SUBAPPLICATION Versuch_405 (* Versuch Array Summe *)
  (* Standard: 61499-2; Description: Copyright (c) 2023 Meisterschulen am Ostbahnhof This program and the accompanying materials are made available under the terms of the Eclipse Public License 2.0 which is available at https://www.eclipse.org/legal/epl-2.0/ SPDX-License-Identifier: EPL-2.0 *)
  (* Version 1.0, 2023-10-23, Franz Höpfinger, Meisterschulen am Ostbahnhof *)
  PACKAGE Versuche;
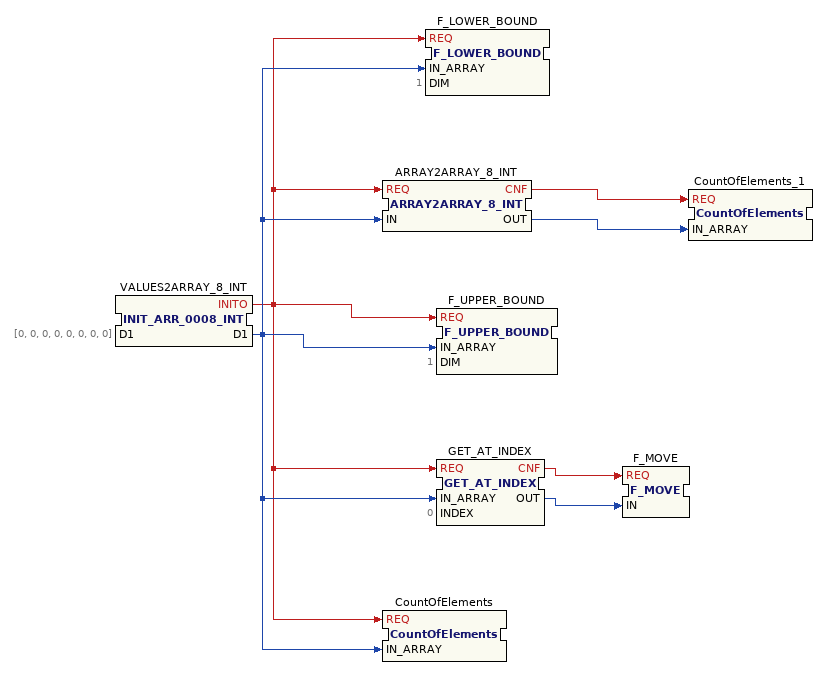
  FBS
    GET_AT_INDEX : eclipse4diac::convert::GET_AT_INDEX(INDEX := 0);
    F_MOVE : iec61131::selection::F_MOVE; {SET_ATTRIBUTE(DataType, INT)}
    CountOfElements : eclipse4diac::convert::CountOfElements;
    F_UPPER_BOUND : eclipse4diac::convert::F_UPPER_BOUND(DIM := 1);
    F_LOWER_BOUND : eclipse4diac::convert::F_LOWER_BOUND(DIM := 1);
    VALUES2ARRAY_8_INT : logiBUS::utils::generate::INIT_ARR_0008_INT(D1 := [0, 0, 0, 0, 0, 0, 0, 0]);
    ARRAY2ARRAY_8_INT : eclipse4diac::convert::ARRAY2ARRAY_8_INT;
    CountOfElements_1 : eclipse4diac::convert::CountOfElements;
  END_FBS
  EVENT_CONNECTIONS
    GET_AT_INDEX.CNF TO F_MOVE.REQ;
    VALUES2ARRAY_8_INT.INITO TO GET_AT_INDEX.REQ;
    VALUES2ARRAY_8_INT.INITO TO CountOfElements.REQ;
    VALUES2ARRAY_8_INT.INITO TO F_LOWER_BOUND.REQ;
    VALUES2ARRAY_8_INT.INITO TO F_UPPER_BOUND.REQ;
    VALUES2ARRAY_8_INT.INITO TO ARRAY2ARRAY_8_INT.REQ;
    ARRAY2ARRAY_8_INT.CNF TO CountOfElements_1.REQ;
  END_CONNECTIONS
  DATA_CONNECTIONS
    GET_AT_INDEX.OUT TO F_MOVE.IN;
    VALUES2ARRAY_8_INT.D1 TO GET_AT_INDEX.IN_ARRAY;
    VALUES2ARRAY_8_INT.D1 TO F_UPPER_BOUND.IN_ARRAY;
    VALUES2ARRAY_8_INT.D1 TO F_LOWER_BOUND.IN_ARRAY;
    VALUES2ARRAY_8_INT.D1 TO CountOfElements.IN_ARRAY;
    VALUES2ARRAY_8_INT.D1 TO ARRAY2ARRAY_8_INT.IN;
    ARRAY2ARRAY_8_INT.OUT TO CountOfElements_1.IN_ARRAY;
  END_CONNECTIONS
END_SUBAPPLICATION
